/// Enumeration of all Cylinder
TYPE E_Cylinder :
(
	eCylinder_Toolselector					:= 0,

	
	// IMPORTANT: last entry
	eCylinder_max
);
END_TYPE

(* stored: Version 1.1.0.1, ProductVersion 3.1.4022.10
   DUT E_Cylinder: Id {05c99de9-f803-4e9f-93b7-a9be9815724f} *)
